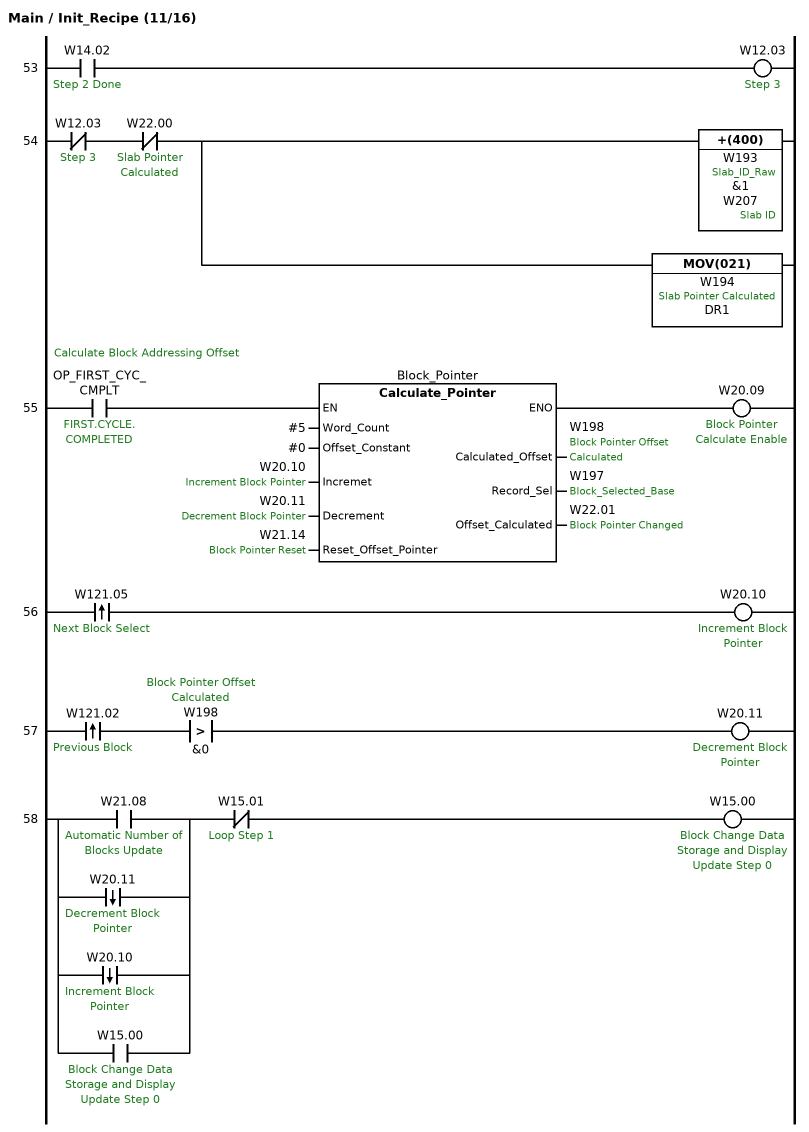
; [picture p24: Main / Init_Recipe, rungs 53-58]
; rung 53
LD W14.02  ; Step 2 Done
OUT W12.03  ; Step 3
; rung 54
LDNOT W12.03  ; Step 3
ANDNOT W22.00  ; Slab Pointer Calculated
+(400) W193 &1 W207  ; Slab_ID_Raw, Slab ID
MOV(021) W194 DR1  ; Slab Pointer Calculated
; rung 55: Calculate Block Addressing Offset
LD OP_FIRST_CYC_CMPLT  ; FIRST.CYCLE.COMPLETED
CALL Block_Pointer : Calculate_Pointer (Word_Count := #5, Offset_Constant := #0, Incremet := W20.10, Decrement := W20.11, Reset_Offset_Pointer := W21.14, Calculated_Offset => W198, Record_Sel => W197, Offset_Calculated => W22.01)  ; Increment Block Pointer, Decrement Block Pointer, Block Pointer Reset, Block Pointer Offset Calculated, Block_Selected_Base, Block Pointer Changed
OUT W20.09  ; Block Pointer Calculate Enable
; rung 56
@LD W121.05  ; Next Block Select
OUT W20.10  ; Increment Block Pointer
; rung 57
@LD W121.02  ; Previous Block
AND>(320) W198 &0  ; Block Pointer Offset Calculated
OUT W20.11  ; Decrement Block Pointer
; rung 58
LD W21.08  ; Automatic Number of Blocks Update
%OR W20.11  ; Decrement Block Pointer
%OR W20.10  ; Increment Block Pointer
OR W15.00  ; Block Change Data Storage and Display Update Step 0
ANDNOT W15.01  ; Loop Step 1
OUT W15.00  ; Block Change Data Storage and Display Update Step 0

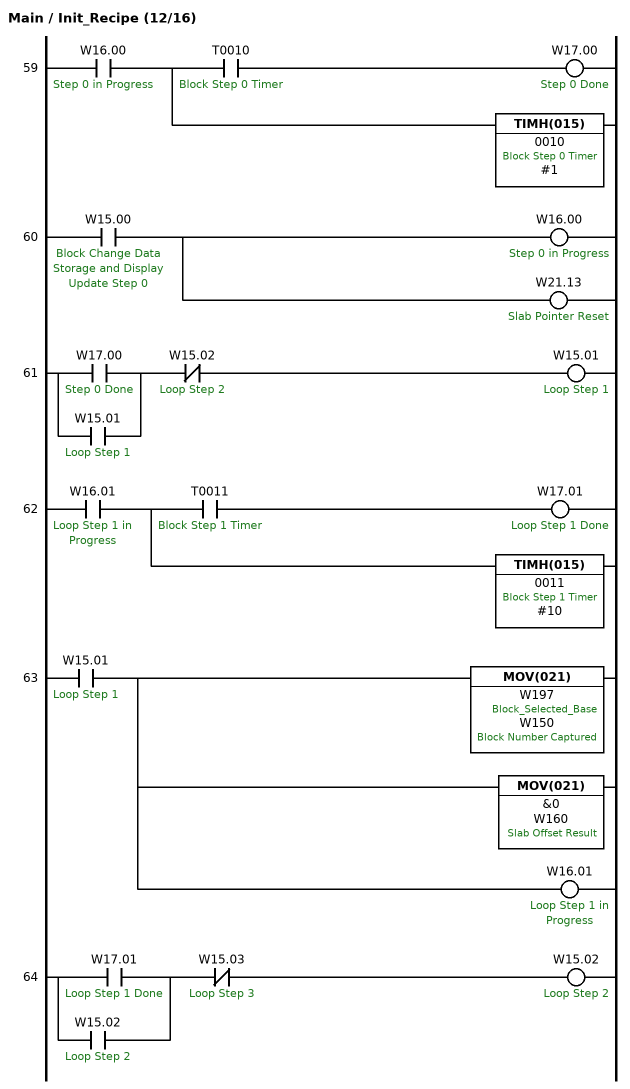
; rung 59
LD W16.00  ; Step 0 in Progress
OUT TR0
AND T0010  ; Block Step 0 Timer
OUT W17.00  ; Step 0 Done
LD TR0
TIMH(015) 0010 #1  ; Block Step 0 Timer
; rung 60
LD W15.00  ; Block Change Data Storage and Display Update Step 0
OUT W16.00  ; Step 0 in Progress
OUT W21.13  ; Slab Pointer Reset
; rung 61
LD W17.00  ; Step 0 Done
OR W15.01  ; Loop Step 1
ANDNOT W15.02  ; Loop Step 2
OUT W15.01  ; Loop Step 1
; rung 62
LD W16.01  ; Loop Step 1 in Progress
OUT TR0
AND T0011  ; Block Step 1 Timer
OUT W17.01  ; Loop Step 1 Done
LD TR0
TIMH(015) 0011 #10  ; Block Step 1 Timer
; rung 63
LD W15.01  ; Loop Step 1
MOV(021) W197 W150  ; Block_Selected_Base, Block Number Captured
MOV(021) &0 W160  ; Slab Offset Result
OUT W16.01  ; Loop Step 1 in Progress
; rung 64
LD W17.01  ; Loop Step 1 Done
OR W15.02  ; Loop Step 2
ANDNOT W15.03  ; Loop Step 3
OUT W15.02  ; Loop Step 2

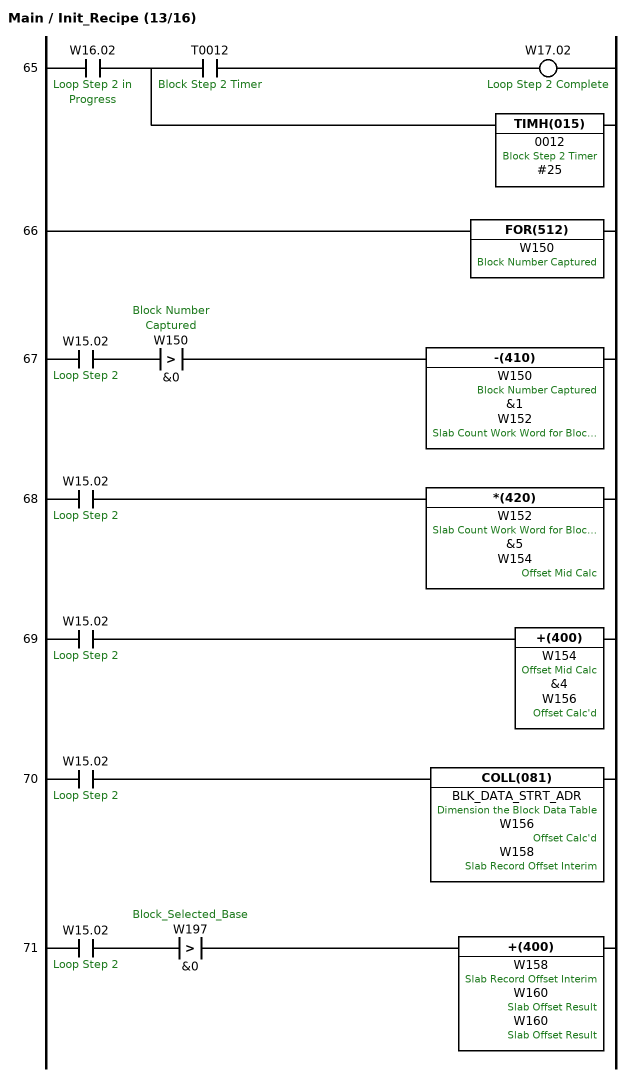
; rung 65
LD W16.02  ; Loop Step 2 in Progress
OUT TR0
AND T0012  ; Block Step 2 Timer
OUT W17.02  ; Loop Step 2 Complete
LD TR0
TIMH(015) 0012 #25  ; Block Step 2 Timer
; rung 66
FOR(512) W150  ; Block Number Captured
; rung 67
LD W15.02  ; Loop Step 2
AND>(320) W150 &0  ; Block Number Captured
-(410) W150 &1 W152  ; Block Number Captured, Slab Count Work Word for Block Pointer
; rung 68
LD W15.02  ; Loop Step 2
*(420) W152 &5 W154  ; Slab Count Work Word for Block Pointer, Offset Mid Calc
; rung 69
LD W15.02  ; Loop Step 2
+(400) W154 &4 W156  ; Offset Mid Calc, Offset Calc'd
; rung 70
LD W15.02  ; Loop Step 2
COLL(081) BLK_DATA_STRT_ADR W156 W158  ; Dimension the Block Data Table, Offset Calc'd, Slab Record Offset Interim
; rung 71
LD W15.02  ; Loop Step 2
AND>(320) W197 &0  ; Block_Selected_Base
+(400) W158 W160 W160  ; Slab Record Offset Interim, Slab Offset Result

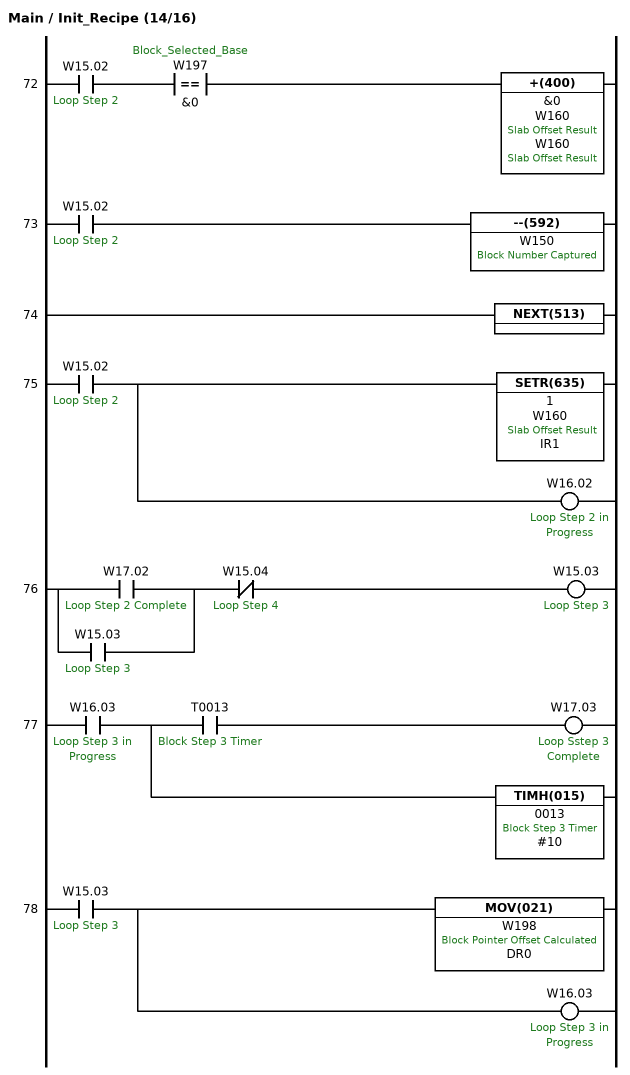
; rung 72
LD W15.02  ; Loop Step 2
AND=(300) W197 &0  ; Block_Selected_Base
+(400) &0 W160 W160  ; Slab Offset Result
; rung 73
LD W15.02  ; Loop Step 2
--(592) W150  ; Block Number Captured
; rung 74
NEXT(513)
; rung 75
LD W15.02  ; Loop Step 2
SETR(635) 1 W160 IR1  ; Slab Offset Result
OUT W16.02  ; Loop Step 2 in Progress
; rung 76
LD W17.02  ; Loop Step 2 Complete
OR W15.03  ; Loop Step 3
ANDNOT W15.04  ; Loop Step 4
OUT W15.03  ; Loop Step 3
; rung 77
LD W16.03  ; Loop Step 3 in Progress
OUT TR0
AND T0013  ; Block Step 3 Timer
OUT W17.03  ; Loop Sstep 3 Complete
LD TR0
TIMH(015) 0013 #10  ; Block Step 3 Timer
; rung 78
LD W15.03  ; Loop Step 3
MOV(021) W198 DR0  ; Block Pointer Offset Calculated
OUT W16.03  ; Loop Step 3 in Progress

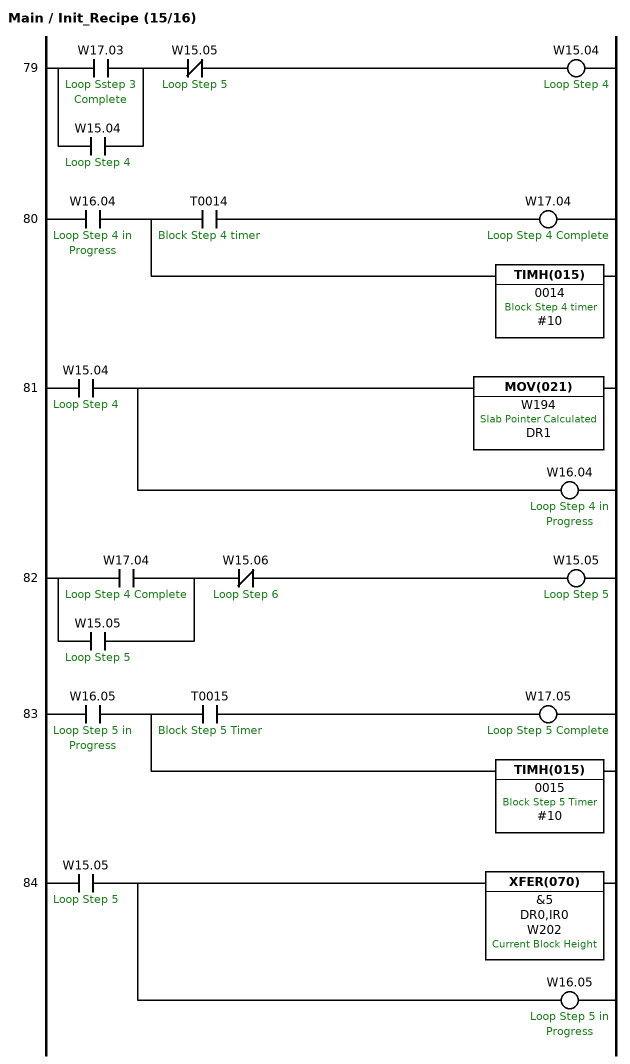
; rung 79
LD W17.03  ; Loop Sstep 3 Complete
OR W15.04  ; Loop Step 4
ANDNOT W15.05  ; Loop Step 5
OUT W15.04  ; Loop Step 4
; rung 80
LD W16.04  ; Loop Step 4 in Progress
OUT TR0
AND T0014  ; Block Step 4 timer
OUT W17.04  ; Loop Step 4 Complete
LD TR0
TIMH(015) 0014 #10  ; Block Step 4 timer
; rung 81
LD W15.04  ; Loop Step 4
MOV(021) W194 DR1  ; Slab Pointer Calculated
OUT W16.04  ; Loop Step 4 in Progress
; rung 82
LD W17.04  ; Loop Step 4 Complete
OR W15.05  ; Loop Step 5
ANDNOT W15.06  ; Loop Step 6
OUT W15.05  ; Loop Step 5
; rung 83
LD W16.05  ; Loop Step 5 in Progress
OUT TR0
AND T0015  ; Block Step 5 Timer
OUT W17.05  ; Loop Step 5 Complete
LD TR0
TIMH(015) 0015 #10  ; Block Step 5 Timer
; rung 84
LD W15.05  ; Loop Step 5
XFER(070) &5 DR0,IR0 W202  ; Current Block Height
OUT W16.05  ; Loop Step 5 in Progress

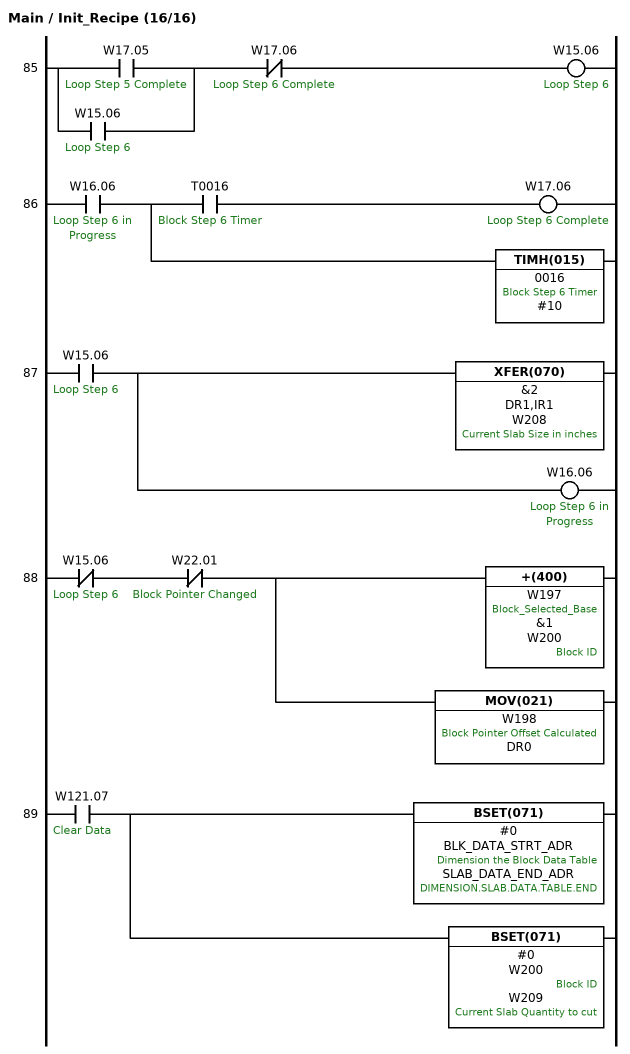
; rung 85
LD W17.05  ; Loop Step 5 Complete
OR W15.06  ; Loop Step 6
ANDNOT W17.06  ; Loop Step 6 Complete
OUT W15.06  ; Loop Step 6
; rung 86
LD W16.06  ; Loop Step 6 in Progress
OUT TR0
AND T0016  ; Block Step 6 Timer
OUT W17.06  ; Loop Step 6 Complete
LD TR0
TIMH(015) 0016 #10  ; Block Step 6 Timer
; rung 87
LD W15.06  ; Loop Step 6
XFER(070) &2 DR1,IR1 W208  ; Current Slab Size in inches
OUT W16.06  ; Loop Step 6 in Progress
; rung 88
LDNOT W15.06  ; Loop Step 6
ANDNOT W22.01  ; Block Pointer Changed
+(400) W197 &1 W200  ; Block_Selected_Base, Block ID
MOV(021) W198 DR0  ; Block Pointer Offset Calculated
; rung 89
LD W121.07  ; Clear Data
BSET(071) #0 BLK_DATA_STRT_ADR SLAB_DATA_END_ADR  ; Dimension the Block Data Table, DIMENSION.SLAB.DATA.TABLE.END
BSET(071) #0 W200 W209  ; Block ID, Current Slab Quantity to cut

### Section Init_Message_Display

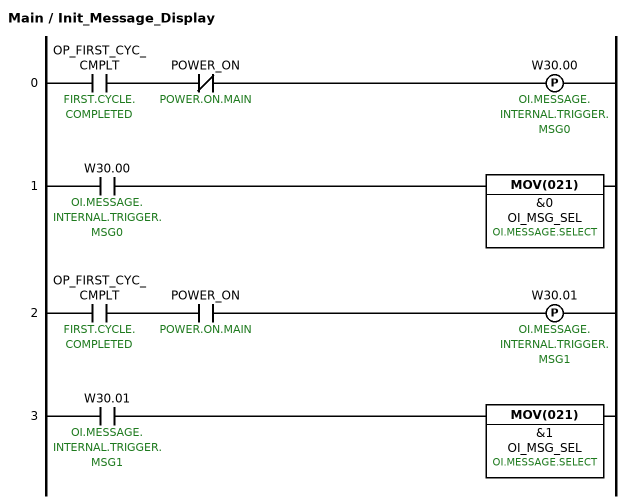
; rung 0
LD OP_FIRST_CYC_CMPLT  ; FIRST.CYCLE.COMPLETED
ANDNOT POWER_ON  ; POWER.ON.MAIN
DIFU(013) W30.00  ; OI.MESSAGE.INTERNAL.TRIGGER.MSG0
; rung 1
LD W30.00  ; OI.MESSAGE.INTERNAL.TRIGGER.MSG0
MOV(021) &0 OI_MSG_SEL  ; OI.MESSAGE.SELECT
; rung 2
LD OP_FIRST_CYC_CMPLT  ; FIRST.CYCLE.COMPLETED
AND POWER_ON  ; POWER.ON.MAIN
DIFU(013) W30.01  ; OI.MESSAGE.INTERNAL.TRIGGER.MSG1
; rung 3
LD W30.01  ; OI.MESSAGE.INTERNAL.TRIGGER.MSG1
MOV(021) &1 OI_MSG_SEL  ; OI.MESSAGE.SELECT

### Section Init_Alarm_Display

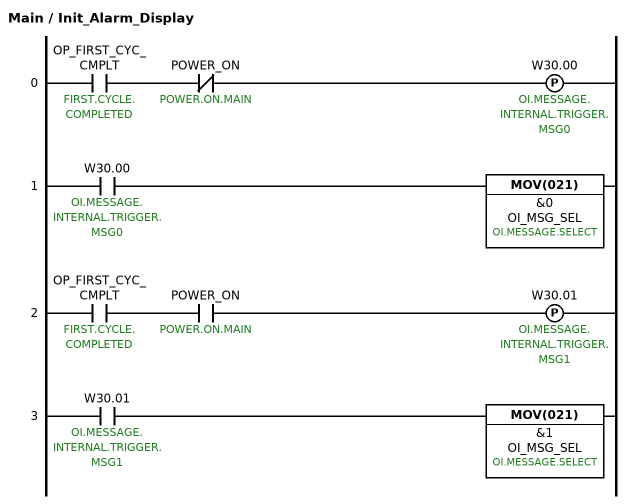
; rung 0
LD OP_FIRST_CYC_CMPLT  ; FIRST.CYCLE.COMPLETED
ANDNOT POWER_ON  ; POWER.ON.MAIN
DIFU(013) W30.00  ; OI.MESSAGE.INTERNAL.TRIGGER.MSG0
; rung 1
LD W30.00  ; OI.MESSAGE.INTERNAL.TRIGGER.MSG0
MOV(021) &0 OI_MSG_SEL  ; OI.MESSAGE.SELECT
; rung 2
LD OP_FIRST_CYC_CMPLT  ; FIRST.CYCLE.COMPLETED
AND POWER_ON  ; POWER.ON.MAIN
DIFU(013) W30.01  ; OI.MESSAGE.INTERNAL.TRIGGER.MSG1
; rung 3
LD W30.01  ; OI.MESSAGE.INTERNAL.TRIGGER.MSG1
MOV(021) &1 OI_MSG_SEL  ; OI.MESSAGE.SELECT

### Section END

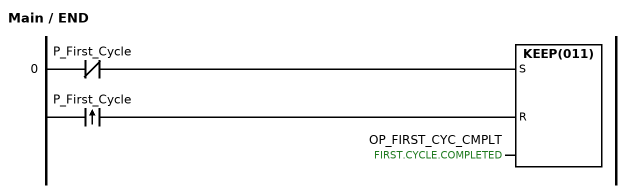
; rung 0
LDNOT P_First_Cycle
@LD P_First_Cycle
KEEP(011) OP_FIRST_CYC_CMPLT  ; FIRST.CYCLE.COMPLETED
; rung 1
END(001)

## Function block Calculate_Pointer
VAR_INPUT
  Word_Count : INT;  (* Number of Words per Record *)
  Offset_Constant : INT;  (* Constant Offset Vaule *)
  Incremet : BOOL;
  Decrement : BOOL;
  Reset_Offset_Pointer : BOOL;  (* Reset Offset and Record Pointers *)
END_VAR
VAR_OUTPUT
  Calculated_Offset : INT;  (* Calculated Offset value *)
  Record_Sel : INT;
  Offset_Calculated : BOOL;  (* Indicates when Offset has been recalculated *)
END_VAR
VAR
  Internal_Count : INT;
  Internal_Calculated_Offset : DINT;
  Internal_Offset_Updated : BOOL;  (* Indicates and update of the offset for use internally. *)
  Internal_Offset_Constant_Compare : INT;  (* Comparison Internal Constant used to trigger a recalulation of the Pointer *)
  Offset_Constant_Changed : BOOL;
  Offset_Calculated_Hold : BOOL;  (* Allow one full scan cycle to complete for the output on time. *)
  TIM100 : BOOL;
END_VAR

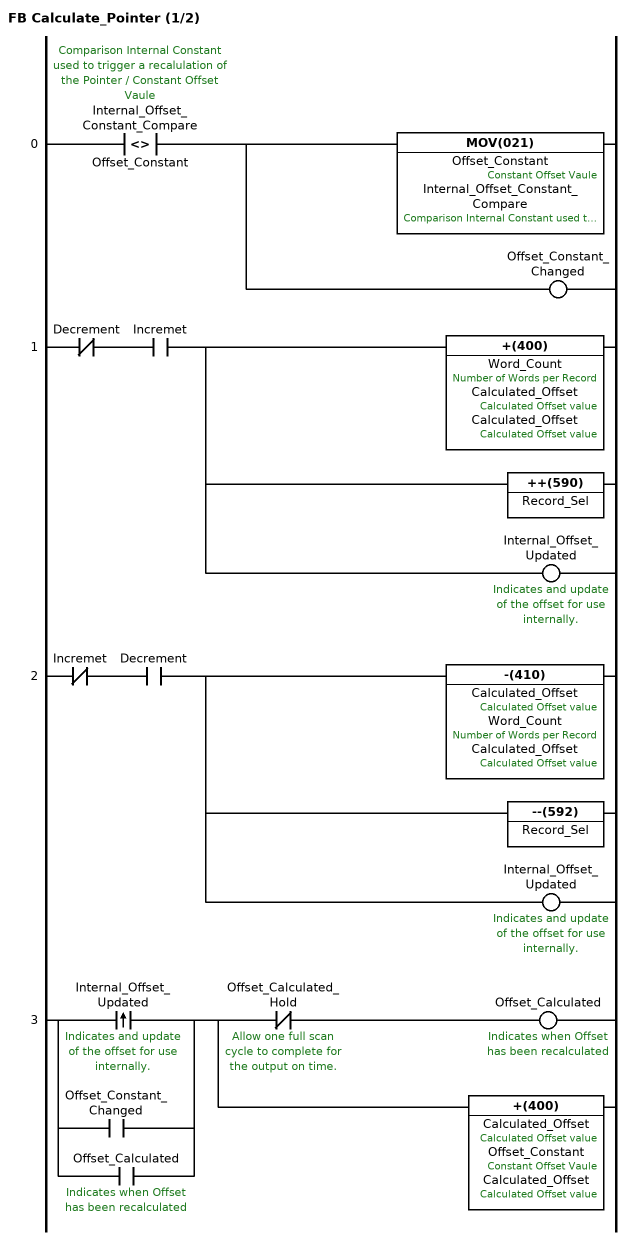
; rung 0
LD<>(305) Internal_Offset_Constant_Compare Offset_Constant  ; Comparison Internal Constant used to trigger a recalulation of the Pointer, Constant Offset Vaule
MOV(021) Offset_Constant Internal_Offset_Constant_Compare  ; Constant Offset Vaule, Comparison Internal Constant used to trigger a recalulation of the Pointer
OUT Offset_Constant_Changed
; rung 1
LDNOT Decrement
AND Incremet
+(400) Word_Count Calculated_Offset Calculated_Offset  ; Number of Words per Record, Calculated Offset value
++(590) Record_Sel
OUT Internal_Offset_Updated  ; Indicates and update of the offset for use internally.
; rung 2
LDNOT Incremet
AND Decrement
-(410) Calculated_Offset Word_Count Calculated_Offset  ; Calculated Offset value, Number of Words per Record
--(592) Record_Sel
OUT Internal_Offset_Updated  ; Indicates and update of the offset for use internally.
; rung 3
@LD Internal_Offset_Updated  ; Indicates and update of the offset for use internally.
OR Offset_Constant_Changed
OR Offset_Calculated  ; Indicates when Offset has been recalculated
OUT TR0
ANDNOT Offset_Calculated_Hold  ; Allow one full scan cycle to complete for the output on time.
OUT Offset_Calculated  ; Indicates when Offset has been recalculated
LD TR0
+(400) Calculated_Offset Offset_Constant Calculated_Offset  ; Calculated Offset value, Constant Offset Vaule

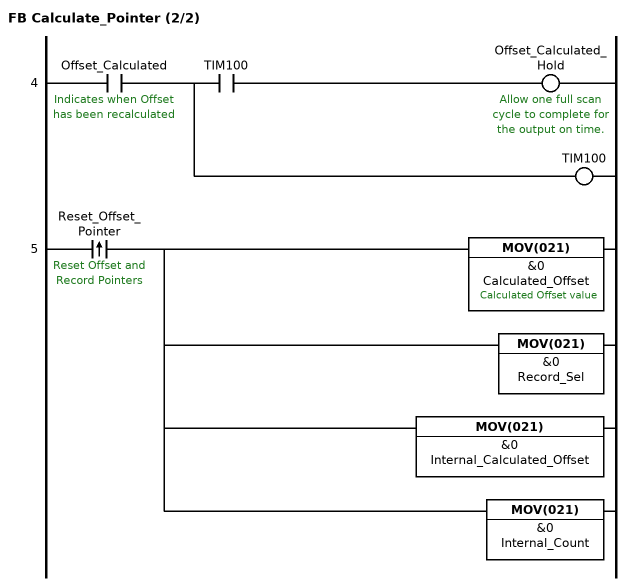
; rung 4
LD Offset_Calculated  ; Indicates when Offset has been recalculated
OUT TR0
AND TIM100
OUT Offset_Calculated_Hold  ; Allow one full scan cycle to complete for the output on time.
LD TR0
OUT TIM100
; rung 5
@LD Reset_Offset_Pointer  ; Reset Offset and Record Pointers
MOV(021) &0 Calculated_Offset  ; Calculated Offset value
MOV(021) &0 Record_Sel
MOV(021) &0 Internal_Calculated_Offset
MOV(021) &0 Internal_Count

## Function block HSC0_INIT
; Initialise HSC Channel Selected
VAR
  Preset : DINT;
END_VAR

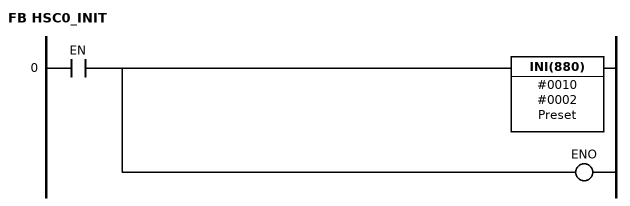
; rung 0
LD EN
INI(880) #0010 #0002 Preset
OUT ENO

## Function block HSC1_INIT
; Initialise HSC Channel Selected
VAR
  Preset : DINT;
END_VAR

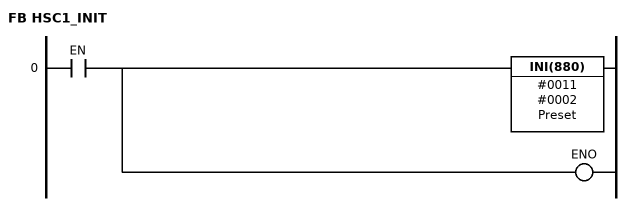
; rung 0
LD EN
INI(880) #0011 #0002 Preset
OUT ENO

## Function block MC_Axis_Home
VAR_INPUT
  INIT : BOOL;  (* Initiate Homing Sequence *)
  REG : BOOL;  (* Registration input *)
  ERR_IN : BOOL;  (* Error monitor *)
END_VAR
VAR_OUTPUT
  CMD_ACTIVE : BOOL;  (* Command is active *)
  CMD_COMPLETE : BOOL;  (* Command is complete *)
  CMD_ERR : BOOL;  (* Command has errored *)
END_VAR
(*Function Block to be used for motion control Homing function*)
ENO:= EN;

## Function block MC_Axis_Jog
VAR_INPUT
  jog_plus : BOOL;  (* Jog in the positive direction *)
  jog_minus : BOOL;  (* Jog in the negative direction *)
  axis_err : BOOL;  (* Drive error status monitor *)
  minus_lim : BOOL;  (* Negative direction limit input *)
  plus_lim : BOOL;  (* Positive direction limit input *)
  JogVelRef : INT;  (* Jog Velocity Reference *)
  Drv_Zero_Spd : BOOL;  (* DRIVE.ZERO.SPEED.INPUT *)
  Brk_En : BOOL;  (* BRAKE.CONTROL.ENABLE *)
END_VAR
VAR_OUTPUT
  jog_plus_cmd : BOOL;  (* Jog in the positive direction command *)
  jog_minus_cmd : BOOL;  (* Jog in the negative direction command *)
  jog_active : BOOL;  (* Jog command is active *)
  jog_err : BOOL;  (* Jog error output *)
  JogVelRefCmd : INT;  (* Jog Velocity Reference Command *)
  Brk_Act : BOOL;  (* BRAKE.CONTROL.ACTIVE.(RELEASE) *)
END_VAR
(*Function Block to be used for motion control jogging function*)
ENO:= EN;
JogVelRefCmd:= JogVelRef;
IF (axis_err = TRUE)THEN jog_err:= TRUE;
	jog_minus_cmd:= FALSE;
	jog_plus_cmd:= FALSE;
	jog_active:= FALSE;
	Brk_Act:= FALSE;
ELSIF(axis_err = FALSE)THEN jog_err:= FALSE;
	IF(jog_plus = TRUE AND jog_minus = FALSE)THEN 
		IF(Brk_En = TRUE) THEN Brk_Act:= TRUE;
			TIMH(TRUE,T20,30);
			IF(T20 = TRUE) THEN jog_plus_cmd:= TRUE;
			END_IF;
		END_IF;
		jog_plus_cmd:= TRUE;
		jog_minus_cmd:= FALSE;
	ELSIF(jog_minus = TRUE AND jog_plus = FALSE)THEN jog_minus_cmd:= TRUE;
		jog_plus_cmd:= FALSE;
	ELSE jog_minus_cmd:= FALSE;
		jog_plus_cmd:= FALSE;
	END_IF;
	IF jog_minus_cmd OR jog_plus_cmd THEN jog_active:= TRUE;
	ELSE jog_active:= FALSE;
	END_IF;
END_IF;

## Function block MC_Axis_Reset
VAR_INPUT
  RST : BOOL;  (* Axis Reset Command *)
END_VAR
VAR_OUTPUT
  RST_REQ : BOOL;  (* Reset Request *)
END_VAR
(* Reset errored Drive*)
ENO:= EN;
IF(RST) THEN RST_REQ:= TRUE;
ELSE RST_REQ:= FALSE;
END_IF;

## Function block Mode_Ind
VAR_INPUT
  MODE_0 : BOOL;  (* Mode 0 *)
  MODE_1 : BOOL;  (* Mode 1 *)
  ERR_IN : BOOL;  (* Error In *)
  START_IN : BOOL;
  STOP_IN : BOOL;
  CYCLE_IN : BOOL;  (* In cycle input *)
  HOME_ACT : BOOL;  (* Homing is active input *)
END_VAR
VAR_OUTPUT
  IND_0 : BOOL;
  IND_1 : BOOL;
END_VAR
ENO:= EN;
IF (MODE_0) THEN IND_1:= FALSE; 
	IF (ERR_IN) THEN 
		IND_0:= EN AND P_0_1s;
	ELSIF (HOME_ACT) THEN IND_0:= EN AND P_1s;
	ELSE IND_0:= TRUE;
	END_IF;
ELSIF (MODE_1) THEN IND_0:= FALSE;
	IF (ERR_IN) THEN
		IND_1:= EN AND P_0_1s;
	ELSIF (START_IN AND NOT CYCLE_IN) THEN IND_1:= EN AND P_0_2s;
	ELSIF (STOP_IN AND CYCLE_IN) THEN IND_1:= EN AND P_0_2s;
	ELSIF(CYCLE_IN AND NOT START_IN AND NOT STOP_IN) THEN IND_1:= TRUE;
	ELSE IND_1:= EN AND P_1min;
	END_IF;
END_IF;

## Function block Op_2_State
VAR_INPUT
  op_state : BOOL;  (* Control Power Status Input from process. *)
END_VAR
VAR_OUTPUT
  op_err : BOOL;  (* Control Power Error Status for User Program use. *)
END_VAR
IF (op_state)THEN 
	ENO := TRUE;
	op_err:= FALSE;
ELSE 
	ENO:=FALSE;
	op_err:= TRUE;
END_IF;

## Function block Op_Message
VAR_INPUT
  Message_Select : INT;  (* Select Message to Display *)
  Message_Trigger : BOOL;  (* Trigger Message Change *)
  Message_Colour : INT;  (* Select Message Text Colour *)
END_VAR
VAR_OUTPUT
  Message_Display : INT;  (* Message to display *)
  Message_Colour_Set : INT;  (* Message Colour to Display *)
END_VAR
IF(Message_Trigger)THEN
	Message_Display:= Message_Select;
	Message_Colour_Set:= Message_Colour;
END_IF;

## Function block Op_Mode_Sel
VAR_INPUT
  Mode_Sel : BOOL;  (* Input to Select Mode *)
END_VAR
VAR_OUTPUT
  Mode_1 : BOOL;  (* Mode 1 selected *)
  Mode_0 : BOOL;  (* Mode 0 selected *)
END_VAR
IF(Mode_Sel) THEN Mode_1:= TRUE;
	Mode_0:= FALSE;
ELSE Mode_1:= FALSE;
	Mode_0:= TRUE;
END_IF;
ENO:= TRUE;